   1:  PR[GP1:91,1] = PR[GP1:90,1] + -46.581;
   1:  PR[GP1:91,2] = PR[GP1:90,2] + 15.215;
   1:L PR[91] 10mm/sec CNT100;
   1:  PR[GP1:91,1] = PR[GP1:90,1] + -48.983;
   1:  PR[GP1:91,2] = PR[GP1:90,2] + -0.010;
   1:L PR[91] 10mm/sec CNT100;
   1:  PR[GP1:91,1] = PR[GP1:90,1] + -48.930;
   1:  PR[GP1:91,2] = PR[GP1:90,2] + -0.388;
   1:L PR[91] 10mm/sec CNT100;
   1:  PR[GP1:91,1] = PR[GP1:90,1] + -46.581;
   1:  PR[GP1:91,2] = PR[GP1:90,2] + -15.223;
   1:L PR[91] 10mm/sec CNT100;
   1:  PR[GP1:91,1] = PR[GP1:90,1] + -46.426;
   1:  PR[GP1:91,2] = PR[GP1:90,2] + -15.573;
   1:L PR[91] 10mm/sec CNT100;
   1:  PR[GP1:91,1] = PR[GP1:90,1] + -39.607;
   1:  PR[GP1:91,2] = PR[GP1:90,2] + -28.956;
   1:L PR[91] 10mm/sec CNT100;
   1:  PR[GP1:91,1] = PR[GP1:90,1] + -39.363;
   1:  PR[GP1:91,2] = PR[GP1:90,2] + -29.250;
   1:L PR[91] 10mm/sec CNT100;
   1:  PR[GP1:91,1] = PR[GP1:90,1] + -28.739;
   1:  PR[GP1:91,2] = PR[GP1:90,2] + -39.874;
   1:L PR[91] 10mm/sec CNT100;
   1:  PR[GP1:91,1] = PR[GP1:90,1] + -28.470;
   1:  PR[GP1:91,2] = PR[GP1:90,2] + -40.065;
   1:L PR[91] 10mm/sec CNT100;
   1:  PR[GP1:91,1] = PR[GP1:90,1] + -15.079;
   1:  PR[GP1:91,2] = PR[GP1:90,2] + -46.888;
   1:L PR[91] 10mm/sec CNT100;
   1:  PR[GP1:91,1] = PR[GP1:90,1] + -14.781;
   1:  PR[GP1:91,2] = PR[GP1:90,2] + -47.003;
   1:L PR[91] 10mm/sec CNT100;
   1:  PR[GP1:91,1] = PR[GP1:90,1] + -14.424;
   1:  PR[GP1:91,2] = PR[GP1:90,2] + -47.047;
   1:L PR[91] 10mm/sec CNT100;
   1:  PR[GP1:91,1] = PR[GP1:90,1] + 0.420;
   1:  PR[GP1:91,2] = PR[GP1:90,2] + -49.399;
   1:L PR[91] 10mm/sec CNT100;
   1:  PR[GP1:91,1] = PR[GP1:90,1] + 0.747;
   1:  PR[GP1:91,2] = PR[GP1:90,2] + -49.358;
   1:L PR[91] 10mm/sec CNT100;
   1:  PR[GP1:91,1] = PR[GP1:90,1] + 15.592;
   1:  PR[GP1:91,2] = PR[GP1:90,2] + -47.007;
   1:L PR[91] 10mm/sec CNT100;
   1:  PR[GP1:91,1] = PR[GP1:90,1] + 15.899;
   1:  PR[GP1:91,2] = PR[GP1:90,2] + -46.888;
   1:L PR[91] 10mm/sec CNT100;
   1:  PR[GP1:91,1] = PR[GP1:90,1] + 29.291;
   1:  PR[GP1:91,2] = PR[GP1:90,2] + -40.065;
   1:L PR[91] 10mm/sec CNT100;
   1:  PR[GP1:91,1] = PR[GP1:90,1] + 29.560;
   1:  PR[GP1:91,2] = PR[GP1:90,2] + -39.874;
   1:L PR[91] 10mm/sec CNT100;
   1:  PR[GP1:91,1] = PR[GP1:90,1] + 40.184;
   1:  PR[GP1:91,2] = PR[GP1:90,2] + -29.250;
   1:L PR[91] 10mm/sec CNT100;
   1:  PR[GP1:91,1] = PR[GP1:90,1] + 40.428;
   1:  PR[GP1:91,2] = PR[GP1:90,2] + -28.956;
   1:L PR[91] 10mm/sec CNT100;
   1:  PR[GP1:91,1] = PR[GP1:90,1] + 47.247;
   1:  PR[GP1:91,2] = PR[GP1:90,2] + -15.573;
   1:L PR[91] 10mm/sec CNT100;
   1:  PR[GP1:91,1] = PR[GP1:90,1] + 47.401;
   1:  PR[GP1:91,2] = PR[GP1:90,2] + -15.223;
   1:L PR[91] 10mm/sec CNT100;
   1:  PR[GP1:91,1] = PR[GP1:90,1] + 49.803;
   1:  PR[GP1:91,2] = PR[GP1:90,2] + -0.004;
   1:L PR[91] 10mm/sec CNT100;
   1:  PR[GP1:91,1] = PR[GP1:90,1] + 47.401;
   1:  PR[GP1:91,2] = PR[GP1:90,2] + 15.215;
   1:L PR[91] 10mm/sec CNT100;
   1:  PR[GP1:91,1] = PR[GP1:90,1] + 47.247;
   1:  PR[GP1:91,2] = PR[GP1:90,2] + 15.564;
   1:L PR[91] 10mm/sec CNT100;
   1:  PR[GP1:91,1] = PR[GP1:90,1] + 40.428;
   1:  PR[GP1:91,2] = PR[GP1:90,2] + 28.947;
   1:L PR[91] 10mm/sec CNT100;
   1:  PR[GP1:91,1] = PR[GP1:90,1] + 40.184;
   1:  PR[GP1:91,2] = PR[GP1:90,2] + 29.241;
   1:L PR[91] 10mm/sec CNT100;
   1:  PR[GP1:91,1] = PR[GP1:90,1] + 29.560;
   1:  PR[GP1:91,2] = PR[GP1:90,2] + 39.865;
   1:L PR[91] 10mm/sec CNT100;
   1:  PR[GP1:91,1] = PR[GP1:90,1] + 29.291;
   1:  PR[GP1:91,2] = PR[GP1:90,2] + 40.056;
   1:L PR[91] 10mm/sec CNT100;
   1:  PR[GP1:91,1] = PR[GP1:90,1] + 15.899;
   1:  PR[GP1:91,2] = PR[GP1:90,2] + 46.879;
   1:L PR[91] 10mm/sec CNT100;
   1:  PR[GP1:91,1] = PR[GP1:90,1] + 15.592;
   1:  PR[GP1:91,2] = PR[GP1:90,2] + 46.998;
   1:L PR[91] 10mm/sec CNT100;
   1:  PR[GP1:91,1] = PR[GP1:90,1] + 0.747;
   1:  PR[GP1:91,2] = PR[GP1:90,2] + 49.349;
   1:L PR[91] 10mm/sec CNT100;
   1:  PR[GP1:91,1] = PR[GP1:90,1] + 0.410;
   1:  PR[GP1:91,2] = PR[GP1:90,2] + 49.391;
   1:L PR[91] 10mm/sec CNT100;
   1:  PR[GP1:91,1] = PR[GP1:90,1] + 0.073;
   1:  PR[GP1:91,2] = PR[GP1:90,2] + 49.349;
   1:L PR[91] 10mm/sec CNT100;
   1:  PR[GP1:91,1] = PR[GP1:90,1] + -14.771;
   1:  PR[GP1:91,2] = PR[GP1:90,2] + 46.998;
   1:L PR[91] 10mm/sec CNT100;
   1:  PR[GP1:91,1] = PR[GP1:90,1] + -15.079;
   1:  PR[GP1:91,2] = PR[GP1:90,2] + 46.879;
   1:L PR[91] 10mm/sec CNT100;
   1:  PR[GP1:91,1] = PR[GP1:90,1] + -28.470;
   1:  PR[GP1:91,2] = PR[GP1:90,2] + 40.056;
   1:L PR[91] 10mm/sec CNT100;
   1:  PR[GP1:91,1] = PR[GP1:90,1] + -28.739;
   1:  PR[GP1:91,2] = PR[GP1:90,2] + 39.865;
   1:L PR[91] 10mm/sec CNT100;
   1:  PR[GP1:91,1] = PR[GP1:90,1] + -39.363;
   1:  PR[GP1:91,2] = PR[GP1:90,2] + 29.241;
   1:L PR[91] 10mm/sec CNT100;
   1:  PR[GP1:91,1] = PR[GP1:90,1] + -39.607;
   1:  PR[GP1:91,2] = PR[GP1:90,2] + 28.947;
   1:L PR[91] 10mm/sec CNT100;
   1:  PR[GP1:91,1] = PR[GP1:90,1] + -46.426;
   1:  PR[GP1:91,2] = PR[GP1:90,2] + 15.564;
   1:L PR[91] 10mm/sec CNT100;
   1:  PR[GP1:91,1] = PR[GP1:90,1] + -46.581;
   1:  PR[GP1:91,2] = PR[GP1:90,2] + 15.215;
   1:L PR[91] 10mm/sec CNT100;
   1:  PR[GP1:91,1] = PR[GP1:90,1] + -48.983;
   1:  PR[GP1:91,2] = PR[GP1:90,2] + -0.010;
   1:L PR[91] 10mm/sec CNT100;
   1:  PR[GP1:91,1] = PR[GP1:90,1] + -48.930;
   1:  PR[GP1:91,2] = PR[GP1:90,2] + -0.388;
   1:L PR[91] 10mm/sec CNT100;
   1:  PR[GP1:91,1] = PR[GP1:90,1] + -46.581;
   1:  PR[GP1:91,2] = PR[GP1:90,2] + -15.223;
   1:L PR[91] 10mm/sec CNT100;
   1:  PR[GP1:91,1] = PR[GP1:90,1] + -46.426;
   1:  PR[GP1:91,2] = PR[GP1:90,2] + -15.573;
   1:L PR[91] 10mm/sec CNT100;
   1:  PR[GP1:91,1] = PR[GP1:90,1] + -39.607;
   1:  PR[GP1:91,2] = PR[GP1:90,2] + -28.956;
   1:L PR[91] 10mm/sec CNT100;
   1:  PR[GP1:91,1] = PR[GP1:90,1] + -39.363;
   1:  PR[GP1:91,2] = PR[GP1:90,2] + -29.250;
   1:L PR[91] 10mm/sec CNT100;
   1:  PR[GP1:91,1] = PR[GP1:90,1] + -28.739;
   1:  PR[GP1:91,2] = PR[GP1:90,2] + -39.874;
   1:L PR[91] 10mm/sec CNT100;
   1:  PR[GP1:91,1] = PR[GP1:90,1] + -28.470;
   1:  PR[GP1:91,2] = PR[GP1:90,2] + -40.065;
   1:L PR[91] 10mm/sec CNT100;
   1:  PR[GP1:91,1] = PR[GP1:90,1] + -15.079;
   1:  PR[GP1:91,2] = PR[GP1:90,2] + -46.888;
   1:L PR[91] 10mm/sec CNT100;
   1:  PR[GP1:91,1] = PR[GP1:90,1] + -14.781;
   1:  PR[GP1:91,2] = PR[GP1:90,2] + -47.003;
   1:L PR[91] 10mm/sec CNT100;
   1:  PR[GP1:91,1] = PR[GP1:90,1] + -14.424;
   1:  PR[GP1:91,2] = PR[GP1:90,2] + -47.047;
   1:L PR[91] 10mm/sec CNT100;
   1:  PR[GP1:91,1] = PR[GP1:90,1] + 0.420;
   1:  PR[GP1:91,2] = PR[GP1:90,2] + -49.399;
   1:L PR[91] 10mm/sec CNT100;
   1:  PR[GP1:91,1] = PR[GP1:90,1] + 0.747;
   1:  PR[GP1:91,2] = PR[GP1:90,2] + -49.358;
   1:L PR[91] 10mm/sec CNT100;
   1:  PR[GP1:91,1] = PR[GP1:90,1] + 15.592;
   1:  PR[GP1:91,2] = PR[GP1:90,2] + -47.007;
   1:L PR[91] 10mm/sec CNT100;
   1:  PR[GP1:91,1] = PR[GP1:90,1] + 15.899;
   1:  PR[GP1:91,2] = PR[GP1:90,2] + -46.888;
   1:L PR[91] 10mm/sec CNT100;
   1:  PR[GP1:91,1] = PR[GP1:90,1] + 29.291;
   1:  PR[GP1:91,2] = PR[GP1:90,2] + -40.065;
   1:L PR[91] 10mm/sec CNT100;
   1:  PR[GP1:91,1] = PR[GP1:90,1] + 29.560;
   1:  PR[GP1:91,2] = PR[GP1:90,2] + -39.874;
   1:L PR[91] 10mm/sec CNT100;
   1:  PR[GP1:91,1] = PR[GP1:90,1] + 40.184;
   1:  PR[GP1:91,2] = PR[GP1:90,2] + -29.250;
   1:L PR[91] 10mm/sec CNT100;
   1:  PR[GP1:91,1] = PR[GP1:90,1] + 40.428;
   1:  PR[GP1:91,2] = PR[GP1:90,2] + -28.956;
   1:L PR[91] 10mm/sec CNT100;
   1:  PR[GP1:91,1] = PR[GP1:90,1] + 47.247;
   1:  PR[GP1:91,2] = PR[GP1:90,2] + -15.573;
   1:L PR[91] 10mm/sec CNT100;
   1:  PR[GP1:91,1] = PR[GP1:90,1] + 47.401;
   1:  PR[GP1:91,2] = PR[GP1:90,2] + -15.223;
   1:L PR[91] 10mm/sec CNT100;
   1:  PR[GP1:91,1] = PR[GP1:90,1] + 49.803;
   1:  PR[GP1:91,2] = PR[GP1:90,2] + -0.004;
   1:L PR[91] 10mm/sec CNT100;
   1:  PR[GP1:91,1] = PR[GP1:90,1] + 47.401;
   1:  PR[GP1:91,2] = PR[GP1:90,2] + 15.215;
   1:L PR[91] 10mm/sec CNT100;
   1:  PR[GP1:91,1] = PR[GP1:90,1] + 47.247;
   1:  PR[GP1:91,2] = PR[GP1:90,2] + 15.564;
   1:L PR[91] 10mm/sec CNT100;
   1:  PR[GP1:91,1] = PR[GP1:90,1] + 40.428;
   1:  PR[GP1:91,2] = PR[GP1:90,2] + 28.947;
   1:L PR[91] 10mm/sec CNT100;
   1:  PR[GP1:91,1] = PR[GP1:90,1] + 40.184;
   1:  PR[GP1:91,2] = PR[GP1:90,2] + 29.241;
   1:L PR[91] 10mm/sec CNT100;
   1:  PR[GP1:91,1] = PR[GP1:90,1] + 29.560;
   1:  PR[GP1:91,2] = PR[GP1:90,2] + 39.865;
   1:L PR[91] 10mm/sec CNT100;
   1:  PR[GP1:91,1] = PR[GP1:90,1] + 29.291;
   1:  PR[GP1:91,2] = PR[GP1:90,2] + 40.056;
   1:L PR[91] 10mm/sec CNT100;
   1:  PR[GP1:91,1] = PR[GP1:90,1] + 15.899;
   1:  PR[GP1:91,2] = PR[GP1:90,2] + 46.879;
   1:L PR[91] 10mm/sec CNT100;
   1:  PR[GP1:91,1] = PR[GP1:90,1] + 15.592;
   1:  PR[GP1:91,2] = PR[GP1:90,2] + 46.998;
   1:L PR[91] 10mm/sec CNT100;
   1:  PR[GP1:91,1] = PR[GP1:90,1] + 0.747;
   1:  PR[GP1:91,2] = PR[GP1:90,2] + 49.349;
   1:L PR[91] 10mm/sec CNT100;
   1:  PR[GP1:91,1] = PR[GP1:90,1] + 0.410;
   1:  PR[GP1:91,2] = PR[GP1:90,2] + 49.391;
   1:L PR[91] 10mm/sec CNT100;
   1:  CALL HOME_ALL;
/POS
/END
